// TIA Portal project "Modbus" (V19)

(* hardware
DEVICE "ET 200SP station_2"  ET 200SP-Station
   slot 0: "Rack_0"  Rack  6ES5 710-8MAx1
   slot 1: "PLC_1"  CPU 1512SP-1 PN  6ES7 512-1DM03-0AB0  V3.0
      slot 32768: "PROFINET interface_1"  X1
   slot 2: "CM PtP_1"  CM PtP  6ES7 137-6AA01-0BA0  V2.0
      slot 1: "CM PtP_1"  CM PtP Sub
   slot 3: "Server module_1"  Server module  6ES7 193-6PA00-0AA0  V1.1
      slot 1: "Server module_1"  Server module
   slot 127: "BA 2xRJ45"  BA 2xRJ45  6ES7 193-6AR00-0AA0  V0.0
      slot 32769: "Port_1"  X1 P1  6ES7 193-6AR00-0AA0
      slot 32770: "Port_2"  X1 P2  6ES7 193-6AR00-0AA0
*)

// ===== PLC "PLC_1"  CPU 1512SP-1 PN =====

VAR_GLOBAL   // PLC tag table "Default tag table"
   "System_Byte" AT %MB1 : Byte;
   "FirstScan" AT %M1.0 : Bool;
   "DiagStatusUpdate" AT %M1.1 : Bool;
   "AlwaysTRUE" AT %M1.2 : Bool;
   "AlwaysFALSE" AT %M1.3 : Bool;
   "Clock_Byte" AT %MB0 : Byte;
   "Clock_10Hz" AT %M0.0 : Bool;
   "Clock_5Hz" AT %M0.1 : Bool;
   "Clock_2.5Hz" AT %M0.2 : Bool;
   "Clock_2Hz" AT %M0.3 : Bool;
   "Clock_1.25Hz" AT %M0.4 : Bool;
   "Clock_1Hz" AT %M0.5 : Bool;
   "Clock_0.625Hz" AT %M0.6 : Bool;
   "Clock_0.5Hz" AT %M0.7 : Bool;
END_VAR

// folder: ModbusDev

TYPE "udtRequestData"
   STRUCT
      uiMBDevAdress : UInt;
      udiAdressRegister : UDInt;
      uiLengthInWords : UInt := 1;
      usiMode : USInt;
      wDataToSend : Int;
   END_STRUCT;
END_TYPE

// folder: ModbusDev/udtDGT1weight

TYPE "udtDGT1weight"
   STRUCT
      x : Bool;
   END_STRUCT;
END_TYPE

// folder: ModbusDev/udtWobitDE38

TYPE "udtWobitDE38"
   STRUCT
      x : Bool;
   END_STRUCT;
END_TYPE

// folder: Modbus/DB

DATA_BLOCK "fbModbus_DB"   // DB1
{ S7_Optimized_Access := 'FALSE' }
VERSION : 0.1
// stored: InstanceOfName fbModbus
"fbModbus"
BEGIN
END_DATA_BLOCK

DATA_BLOCK "dbDataForRequest"   // DB3
{ S7_Optimized_Access := 'TRUE' }
VERSION : 0.1
   VAR
      arrRequestData : Array[0..3] of "udtRequestData";
   END_VAR
BEGIN
   arrRequestData[0].uiMBDevAdress := 1;
   arrRequestData[1].uiMBDevAdress := 1;
   arrRequestData[0].udiAdressRegister := 40101;
   arrRequestData[1].udiAdressRegister := 40102;
   arrRequestData[2].uiMBDevAdress := 1;
   arrRequestData[3].uiMBDevAdress := 1;
   arrRequestData[3].udiAdressRegister := 40104;
   arrRequestData[2].udiAdressRegister := 40103;
END_DATA_BLOCK

DATA_BLOCK "dbDataRecived"   // DB6
{ S7_Optimized_Access := 'TRUE' }
VERSION : 0.1
   VAR
      data : Array[0..249] of Int;
   END_VAR
BEGIN
END_DATA_BLOCK

// folder: (top level)

ORGANIZATION_BLOCK "Main"   // OB1, LAD, ProgramCycle
TITLE = "Main Program Sweep (Cycle)"
{ S7_Optimized_Access := 'TRUE' }
VERSION : 0.1
   VAR_INPUT
      Initial_Call : Bool;   // Initial call of this OB
      Remanence : Bool;   // =True, if remanent data are available
   END_VAR
BEGIN

REGION Network 1
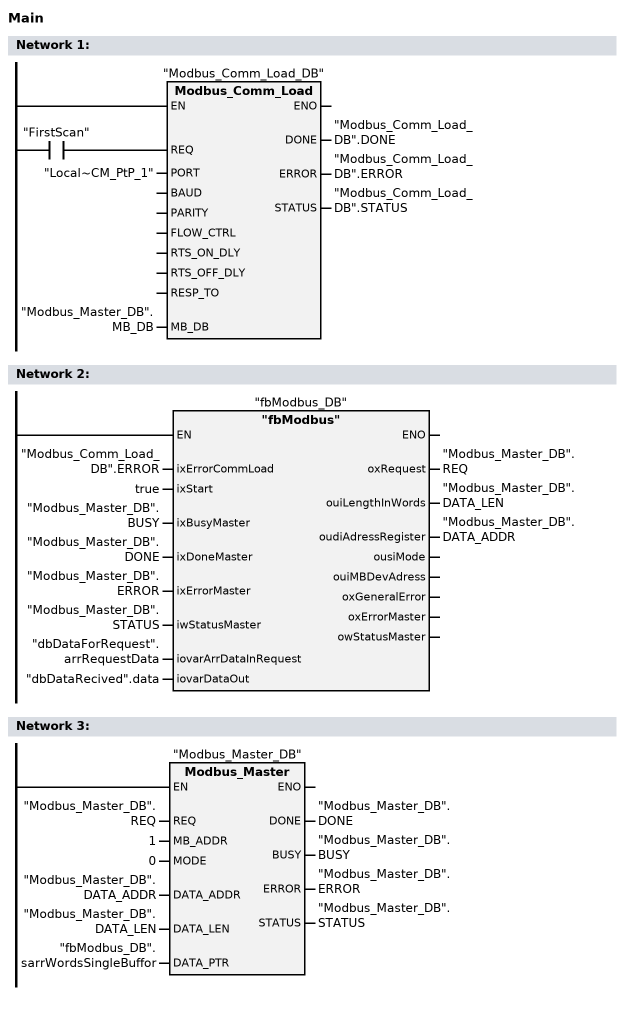
   "Modbus_Comm_Load_DB"(REQ := "FirstScan",   // Modbus_Comm_Load
                         PORT := "Local~CM_PtP_1",
                         MB_DB := "Modbus_Master_DB".MB_DB,
                         DONE => "Modbus_Comm_Load_DB".DONE,
                         ERROR => "Modbus_Comm_Load_DB".ERROR,
                         STATUS => "Modbus_Comm_Load_DB".STATUS);
END_REGION

REGION Network 2
   RUNG wire#powerrail
      "fbModbus_DB"(ixErrorCommLoad := "Modbus_Comm_Load_DB".ERROR, ixStart := true, ixBusyMaster := "Modbus_Master_DB".BUSY, ixDoneMaster := "Modbus_Master_DB".DONE, ixErrorMaster := "Modbus_Master_DB".ERROR, iwStatusMaster := "Modbus_Master_DB".STATUS, iovarArrDataInRequest := "dbDataForRequest".arrRequestData, iovarDataOut := "dbDataRecived".data, oxRequest => "Modbus_Master_DB".REQ, ouiLengthInWords => "Modbus_Master_DB".DATA_LEN, oudiAdressRegister => "Modbus_Master_DB".DATA_ADDR, ousiMode =>, ouiMBDevAdress =>, oxGeneralError =>, oxErrorMaster =>, owStatusMaster =>)
   END_RUNG
   // the same network as SCL:
   "fbModbus_DB"(ixErrorCommLoad := "Modbus_Comm_Load_DB".ERROR,   // "fbModbus"
                 ixStart := true,
                 ixBusyMaster := "Modbus_Master_DB".BUSY,
                 ixDoneMaster := "Modbus_Master_DB".DONE,
                 ixErrorMaster := "Modbus_Master_DB".ERROR,
                 iwStatusMaster := "Modbus_Master_DB".STATUS,
                 iovarArrDataInRequest := "dbDataForRequest".arrRequestData,
                 iovarDataOut := "dbDataRecived".data,
                 oxRequest => "Modbus_Master_DB".REQ,
                 ouiLengthInWords => "Modbus_Master_DB".DATA_LEN,
                 oudiAdressRegister => "Modbus_Master_DB".DATA_ADDR);
END_REGION

REGION Network 3
   "Modbus_Master_DB"(REQ := "Modbus_Master_DB".REQ,   // Modbus_Master
                      MB_ADDR := 1,
                      MODE := 0,
                      DATA_ADDR := "Modbus_Master_DB".DATA_ADDR,
                      DATA_LEN := "Modbus_Master_DB".DATA_LEN,
                      DATA_PTR := "fbModbus_DB".sarrWordsSingleBuffor,
                      DONE => "Modbus_Master_DB".DONE,
                      BUSY => "Modbus_Master_DB".BUSY,
                      ERROR => "Modbus_Master_DB".ERROR,
                      STATUS => "Modbus_Master_DB".STATUS);
END_REGION
END_ORGANIZATION_BLOCK

// folder: Modbus

FUNCTION_BLOCK "fbModbus"   // FB1, SCL
{ S7_Optimized_Access := 'FALSE' }
VERSION : 0.1
   VAR_INPUT
      ixErrorCommLoad : Bool;
      ixStart : Bool;
      ixBusyMaster : Bool;
      ixDoneMaster : Bool;
      ixErrorMaster : Bool;
      iwStatusMaster : Word;
   END_VAR
   VAR_OUTPUT
      oxRequest : Bool;
      ouiLengthInWords : UInt;
      oudiAdressRegister : UDInt;
      ousiMode : USInt;
      ouiMBDevAdress : UInt;
      oxGeneralError : Bool;
      oxErrorMaster : Bool;
      owStatusMaster : Word;
   END_VAR
   VAR_IN_OUT
      iovarArrDataInRequest : Variant;
      iovarDataOut : Variant;
   END_VAR
   VAR
      siStep : Int;
      siStepNew : Int;
      siCounter : Int;
      siStatusErrorMoveBlk1 : Int;
      siStatusErrorMoveBlk2 : Int;
      siStatusSerialize : Int;
      siStatusDeserialize : Int;
      sudtRequestData : "udtRequestData";
      sarrWordsSingleBuffor : Array[0..9] of Int;
      sarrBytesBuffor : Array[0..499] of Byte;
      sarrWordsAllBuffors : Array[0..249] of Int;
      sudiPointerWordsBuffor : UDInt;
      sdiPosSerialize : DInt;
      sdiPosDeserialize : DInt;
      sxGeneralError : Bool;
      instRtrigClock2Hz : R_TRIG;
      instRtrigStart : R_TRIG;
      instRtrigMasterDone : R_TRIG;
      instFtrigMasterDone : F_TRIG;
      instRtrigRequest : R_TRIG;
   END_VAR
   VAR_TEMP
      tudiCountOfDataRequest : UDInt;
      txRequest : Bool;
   END_VAR
BEGIN
   #instRtrigClock2Hz(CLK := "Clock_2Hz");
   #instRtrigStart(CLK := #ixStart);
   #instRtrigMasterDone(CLK := #ixDoneMaster);
   #instFtrigMasterDone(CLK := #ixDoneMaster);

   //get number of elements in Adresses Array
   #tudiCountOfDataRequest := CountOfElements(#iovarArrDataInRequest);

   //main sequencer
   CASE #siStep OF
       0:  // step - init

           // reset all values
           #siStepNew := 0;
           #siCounter := 0;
           #txRequest := false;
           #siStatusErrorMoveBlk1 := 0;
           #siStatusErrorMoveBlk2 := 0;
           #sudiPointerWordsBuffor := 0;

           #sudtRequestData.udiAdressRegister := 0;
           #sudtRequestData.uiLengthInWords := 0;
           #sudtRequestData.uiMBDevAdress := 0;
           #sudtRequestData.usiMode := 0;
           #sudtRequestData.wDataToSend := 0;


           //fill static arrays with zeros
           FILL_BLK(IN := 0,
                    COUNT := 10,
                    OUT => #sarrWordsSingleBuffor[0]);
           FILL_BLK(IN := 0,
                    COUNT := 250,
                    OUT => #sarrWordsAllBuffors[0]);
           FILL_BLK(IN := 0,
                    COUNT := 500,
                    OUT => #sarrBytesBuffor[0]);

           IF #ixStart THEN
               #siStepNew := 10;
           END_IF;

       10:  // Sending request to MB_MASTER
           #txRequest := false;

           //reset temporary single buffer of words
           FILL_BLK(IN := 0,
                    COUNT := 10,
                    OUT => #sarrWordsSingleBuffor[0]);

           //get adress and lenght another element from #inout_varDataAdressAndLength
           #siStatusErrorMoveBlk1 := MOVE_BLK_VARIANT(SRC := #iovarArrDataInRequest,
                                                      SRC_INDEX := #siCounter,
                                                      COUNT := 1,
                                                      DEST_INDEX := 0,
                                                      DEST => #sudtRequestData);


           IF NOT #ixBusyMaster AND #ixStart AND NOT #sxGeneralError AND #instRtrigClock2Hz.Q
               AND #iwStatusMaster <> 16#8200
           THEN
               #siStepNew := 20;
           ELSIF #ixStart = false THEN
               #siStepNew := 0;
           END_IF;

       20: //waiting for DONE from MB_MASTER
           #txRequest := true;


           IF #instRtrigMasterDone.Q AND #ixStart THEN
               #siStepNew := 30;
           ELSIF #iwStatusMaster = 16#8383 THEN
               #siStepNew := 30;
           ELSIF #iwStatusMaster = 16#8200 THEN
               #siStepNew := 10;
           ELSIF #ixStart = false THEN
               #siStepNew := 0;
           END_IF;

       30: // calculate results
           #txRequest := false;

           //move single buffor of words (#arrWordsSingleBuffor) to arrays of buffors (#arrWordsAllBuffors) without empty spaces 
           #siStatusErrorMoveBlk2 := MOVE_BLK_VARIANT(SRC := #sarrWordsSingleBuffor,
                                                      SRC_INDEX := 0,
                                                      COUNT := #sudtRequestData.uiLengthInWords,
                                                      DEST_INDEX := UDINT_TO_DINT(#sudiPointerWordsBuffor),
                                                      DEST => #sarrWordsAllBuffors);

           //serialize array of WORDS #arrWordsAllBuffors to array of BYTES #arrBytesBuffor
           #sdiPosSerialize := 0;
          // #siStatusSerialize:=Serialize(SRC_VARIABLE := #sarrWordsAllBuffors, DEST_ARRAY => #sarrBytesBuffor, POS := #sdiPosSerialize);
           //deserialize array of BYTES #arrBytesBuffor to Struct UDT from inout paramters of function
           #sdiPosDeserialize := 0;
          // #siStatusSerialize := Deserialize(SRC_ARRAY := #sarrBytesBuffor, POS := #sdiPosDeserialize, DEST_VARIABLE => #iovarDataOut);


           IF #ixStart  THEN
               IF #siCounter < #tudiCountOfDataRequest - 1 THEN
                   #siCounter := #siCounter + 1;
                   #sudiPointerWordsBuffor := #sudiPointerWordsBuffor + #sudtRequestData.uiLengthInWords;
               ELSIF #siCounter = #tudiCountOfDataRequest - 1 THEN
                   #siCounter := 0;
                   #sudiPointerWordsBuffor := 0;
               END_IF;
               #siStepNew := 10;
           ELSIF #ixStart = false THEN
               #siStepNew := 0;
           END_IF;
   END_CASE;

   //rewrite number of step
   #siStep := #siStepNew;

   //handle errors
   IF #siStatusErrorMoveBlk1 > 0
       OR #siStatusErrorMoveBlk2 > 0
       OR #siStatusSerialize > 0
       OR #siStatusDeserialize > 0
       OR #ixErrorCommLoad = true THEN
       #sxGeneralError := true;
   ELSE
       #sxGeneralError := false;
   END_IF;

   //rise triger for MB_MASTER request
   #instRtrigRequest(CLK := #txRequest);

   //rewrite outputs
   #oudiAdressRegister := #sudtRequestData.udiAdressRegister;
   #ouiLengthInWords := #sudtRequestData.uiLengthInWords;
   #ouiMBDevAdress := #sudtRequestData.uiMBDevAdress;
   #ousiMode := #sudtRequestData.usiMode;

   #oxRequest := #instRtrigRequest.Q;
   #oxErrorMaster := #ixErrorMaster;
   #owStatusMaster := #iwStatusMaster;
END_FUNCTION_BLOCK